KUKA KRL program: TEST_FREQ.src, TEST_FREQ.dat

--- TEST_FREQ.src ---
&ACCESS RVP
&REL 9
&PARAM TEMPLATE = C:\KRC\Roboter\Template\ExpertVorgabe
&PARAM EDITMASK = *
DEF TEST_FREQ( )
  FREQVAL = GET_FREQ(1, TRUE)

  LOOP
    WAIT SEC 0.1
    FREQVAL = GET_FREQ(1, FALSE)
  ENDLOOP

END

--- TEST_FREQ.dat ---
&ACCESS RVP
&REL 9
&PARAM TEMPLATE = C:\KRC\Roboter\Template\ExpertVorgabe
&PARAM EDITMASK = *
DEFDAT  TEST_FREQ PUBLIC
REAL FREQVAL=10.0308647
ENDDAT
